FUNCTION_BLOCK FB_HVFAStorageSystem EXTENDS FB_SystemContinous
VAR_INPUT
	bLoadingAutomatic : BOOL; //variable to determine if storage is in loading mode
	aTelegramm_WMZ7x0 : ARRAY[1..cMBUS_MaxTelegrams] OF ST_MBus_Data2;
	aTelegramm_WMZx05 : ARRAY[1..cMBUS_MaxTelegrams] OF ST_MBus_Data2;
END_VAR
VAR_OUTPUT
	localState : ST_HVFAStorageState;
END_VAR
VAR
	{attribute 'OPC.UA.DA' := '1'}
	localSetParameters : ST_HVFAStorageSetParameters;
	
	//default parameters
	localDefaultParameters : ST_HVFAStorageSystemDefaultParameters;	

	//storage
	HVFAStorage : FB_HVFAStorage;
	
	//pumps
	PUx05 : FB_PumpGrundfosMagna3; //Magna 3 pump (network side)
	PU7x0 : FB_Pump2Point; //CM pump (storage side)

	//valves
	stSVx05DefaultParameters : ST_MixingValveDefaultParameters := (tTaskCycleTime := GlobalVariables.tCtrlCycleTime_MAIN, tCtrlCycleTime := GlobalVariables.tCtrlCycleTime_MAIN);
	stSVx06DefaultParameters : ST_MixingValveDefaultParameters := (tTaskCycleTime := GlobalVariables.tCtrlCycleTime_MAIN, tCtrlCycleTime := GlobalVariables.tCtrlCycleTime_MAIN);
	stRVx05DefaultParameters : ST_MixingValveDefaultParameters := (tTaskCycleTime := GlobalVariables.tCtrlCycleTime_MAIN, tCtrlCycleTime := GlobalVariables.tCtrlCycleTime_MAIN);
	
	SVx05 : FB_MixingValve := (ST_DefaultParameters := stSVx05DefaultParameters); //discrete inlet valve, valve motor needs continous signal but operates only between extreme positions
	SVx06 : FB_MixingValve := (ST_DefaultParameters := stSVx06DefaultParameters); //discrete outlet valve	, valve motor needs continous signal but operates only between extreme positions
	RVx05 : FB_MixingValve := (ST_DefaultParameters := stRVx05DefaultParameters); //continous mixing valve
	
	//sensors
	WMZ7x0 : FB_MollineC3HeatCounter;
	WMZx05 : FB_MollineC3HeatCounter;
	
	//internal variables
	bSetStatusOn_PUx05 : BOOL;
	bSetStatusOn_PU7x0 : BOOL;
	bSetStatusOn_SVx05 : BOOL;
	fSetPoint_SVx05 : REAL;
	bSetStatusOn_SVx06 : BOOL;
	fSetPoint_SVx06 : REAL;	
	bSetStatusOn_RVx05 : BOOL;
	fSetPoint_RVx05 : REAL;
	fExternalTemperature_RVx05 : REAL;
	nControlMode_RVx05 : E_MixingValveControlMode;
	bLoading : BOOL;
	
	//triggers
	SwitchToLoading : R_TRIG;
	SwitchToUnloading : F_TRIG;
	bFinishedSwitchMode : BOOL := TRUE;
END_VAR

//storage
HVFAStorage(localState => localState);

SelectLoadingMode();
SwitchToLoading(CLK := bLoading);
SwitchToUnloading(CLK := bLoading);

//MAIN must be called before SwitchMode to prevent pump signal chattering (signal is written after SwitchMode function), SwitchMode may only be called if system is on
MAIN();

//disrupt calling SystemFlowControl via MAIN() when mode is switched and call SwitchMode()
IF ((SwitchToLoading.Q OR SwitchToUnloading.Q) OR NOT bFinishedSwitchMode) AND bSetStatusOn THEN
	SwitchMode(bSwitchToLoading := bLoading,
		bFinishedSwitchMode => bFinishedSwitchMode);
END_IF;

//pumps
PUx05.GetState_Profibus();
PUx05(bSetStatusOnAutomatic := bSetStatusOn_PUx05,
	fSetPointAutomatic := 70,
	bAlgorithmPermission := bAlgorithmPermission,
	nControlModeAutomatic := 0);
PUx05.SetState_Profibus();

PU7x0(bSetStatusOnAutomatic := bSetStatusOn_PU7x0,
	bAlgorithmPermission := bAlgorithmPermission);
PU7x0.SetState_BO();

//valves
SVx05.GetState_AI();
SVx05(bSetStatusOnAutomatic := bSetStatusOn_SVx05,
	fSetPointAutomatic := fSetPoint_SVx05,
	bAlgorithmPermission := bAlgorithmPermission,
	nControlModeAutomatic := 0);
SVx05.SetState_AO();

SVx06.GetState_AI();
SVx06(bSetStatusOnAutomatic := bSetStatusOn_SVx06,
	fSetPointAutomatic := fSetPoint_SVx06,
	bAlgorithmPermission := bAlgorithmPermission,
	nControlModeAutomatic := 0);
SVx06.SetState_AO();

RVx05.GetState_AI();
RVx05(bSetStatusOnAutomatic := bSetStatusOn_RVx05,
	fSetPointAutomatic := fSetPoint,
	bAlgorithmPermission := bAlgorithmPermission,
	fTemperatureExternal := fExternalTemperature_RVx05,
	nControlModeAutomatic := 0);
RVx05.SetState_AO();

//insert heat counter telegramm from other task
WMZ7x0(aHeatCounterTelegramm := aTelegramm_WMZ7x0);
WMZx05(aHeatCounterTelegramm := aTelegramm_WMZx05);

IF bLoading = TRUE THEN
	fExternalTemperature_RVx05 := WMZ7x0.fReturnTemperazure;	
ELSE
	fExternalTemperature_RVx05 := WMZx05.fFeedTemperature;
END_IF

METHOD PROTECTED  CheckError : BOOL
VAR_INPUT
END_VAR
VAR_OUTPUT
	bError : BOOL;
END_VAR
VAR
	bError_PUx05 : BOOL;
END_VAR
//check for pump error
bError_PUx05 := PUx05.bError;
END_METHOD

METHOD PROTECTED  Operational : BOOL
VAR_INPUT
END_VAR
VAR_OUTPUT
	bSwitchToWorking : BOOL := FALSE;
END_VAR
//storage pump
bSetStatusOn_PU7x0 := TRUE;

//network pump
bSetStatusOn_PUx05 := TRUE;

//temperature controlling valve
bSetStatusOn_RVx05 := TRUE;

IF PUx05.bStatusOn THEN
	bSwitchToWorking := TRUE;
END_IF
END_METHOD

METHOD PROTECTED  RampDown : BOOL
VAR_INPUT
END_VAR
VAR_OUTPUT
	bRampDownFinished : BOOL := FALSE;
END_VAR
bSetStatusOn_PU7x0 := FALSE;
bSetStatusOn_PUx05 := FALSE;
bSetStatusOn_RVx05 := FALSE;

IF RVx05.fOperatingPoint<20 AND NOT PUx05.bStatusOn THEN
	bRampDownFinished := TRUE;
END_IF
END_METHOD

METHOD PROTECTED  RampUp : BOOL
VAR_INPUT
END_VAR
VAR_OUTPUT
	bRampUpFinished : BOOL := FALSE;
END_VAR
bSetStatusOn_SVx05 := TRUE;
bSetStatusOn_SVx06 := TRUE;

IF bLoading = TRUE THEN
	fSetPoint_SVx05 := 0;
	fSetPoint_SVx06 := 0;
	nControlMode_RVx05 := 2; //cooling mode (heats network)
	fExternalTemperature_RVx05 := WMZ7x0.fReturnTemperazure;	
	IF SVx05.fOperatingPoint<20 AND SVx06.fOperatingPoint<20 THEN
		bRampUpFinished := TRUE;
	END_IF
ELSE
	fSetPoint_SVx05 := 100;
	fSetPoint_SVx06 := 100;
	nControlMode_RVx05 := 1; //heating mode (cools network)
	fExternalTemperature_RVx05 := WMZx05.fFeedTemperature;
	IF SVx05.fOperatingPoint>80 AND SVx06.fOperatingPoint>80 THEN
		bRampUpFinished := TRUE;
	END_IF
END_IF
END_METHOD

METHOD PRIVATE SelectLoadingMode : BOOL
VAR_INPUT
END_VAR
IF control.bManualModeActivated THEN
	bLoading := localSetParameters.bLoadingManual;
ELSIF control.bAlgorithmModeActivated AND bAlgorithmPermission THEN
	bLoading := localSetParameters.bLoadingAlgorithm;
ELSE
	bLoading := bLoadingAutomatic;
END_IF
END_METHOD

METHOD PROTECTED   SetSetPointLimits : BOOL
VAR_INPUT
END_VAR
aSetPointLimits[1] := localDefaultParameters.aSetPointLimitsTemperature[1];
aSetPointLimits[2] := localDefaultParameters.aSetPointLimitsTemperature[2];
END_METHOD

METHOD PROTECTED  SetState : BOOL
VAR_INPUT
END_VAR
VAR_OUTPUT
END_VAR
fOperatingPoint := fExternalTemperature_RVx05;

controlState.bStatusOn := bSetStatusOn;
setPointState.aSetPointLimits := aSetPointLimits;
setPointState.fSetPoint := fSetPoint;
setPointState.fOperatingPoint := fOperatingPoint;
setPointState.sSetPointUnit := 'degreeC';
setPointState.sOperatingPointUnit := 'degreeC';
END_METHOD

PROPERTY ST_DefaultParameters : REFERENCE TO ST_HVFAStorageSystemDefaultParameters
SET
localDefaultParameters := ST_DefaultParameters;
END_SET
END_PROPERTY

METHOD PRIVATE SwitchMode : BOOL
VAR_INPUT
	bSwitchToLoading : BOOL; //if false switch to cooling
END_VAR
VAR_OUTPUT
	bFinishedSwitchMode : BOOL := FALSE;
END_VAR
VAR_INST
	bRampDownFinished : BOOL := FALSE;
END_VAR
//check system state
IF bRampDownFinished THEN
	IF bSwitchToLoading THEN
		fSetPoint_SVx05 := 0;
		fSetPoint_SVx06 := 0;
		nControlMode_RVx05 := 2; //cooling mode (heats network)	
		IF SVx05.fOperatingPoint<20 AND SVx06.fOperatingPoint<20 THEN
			//reset instant variable and switch on pump
			bRampDownFinished := FALSE;			
			bFinishedSwitchMode := TRUE;
			bSetStatusOn_PUx05 := TRUE;
		END_IF
		
	ELSE
		fSetPoint_SVx05 := 100;
		fSetPoint_SVx06 := 100;
		nControlMode_RVx05 := 1; //cooling mode (heats network)	
		IF SVx05.fOperatingPoint>80 AND SVx06.fOperatingPoint>80 THEN
			//reset instant variable and switch on pump
			bRampDownFinished := FALSE;			
			bFinishedSwitchMode := TRUE;
			bSetStatusOn_PUx05 := TRUE;
		END_IF
	END_IF
ELSE
	bSetStatusOn_PUx05 := FALSE;
	IF NOT PUx05.bStatusOn THEN
		bRampDownFinished := TRUE;
	END_IF
END_IF
END_METHOD

METHOD PROTECTED  Working : BOOL
VAR_INPUT
END_VAR
VAR_OUTPUT
	bSwitchToOperational : BOOL := FALSE;
END_VAR
//empty method
END_METHOD

END_FUNCTION_BLOCK

(* stored: Version 1.1.0.1, ProductVersion 3.1.4024.10
   POU FB_HVFAStorageSystem: Id {5fa1e97c-987f-49c1-82cf-2ddae1379d7b}, SpecialFunc None
   Method CheckError: Id {0a750c43-7566-4b1a-a185-b01eaf088ced}
   Method Operational: Id {38ce29c5-a9cb-42f6-b2da-f6e767b8efb9}
   Method RampDown: Id {035f2f79-06b9-4677-b822-1118600ad0da}
   Method RampUp: Id {0ce76782-d529-4b5d-8974-d96ba13ac874}
   Method SelectLoadingMode: Id {324f0df5-410b-4639-a772-5eb1aaf75a71}
   Method SetSetPointLimits: Id {f04c6bfe-2c3e-49d6-a8c4-445113c91ff8}
   Method SetState: Id {e91ff025-34ce-4425-84b2-ec422191accc}
   Property ST_DefaultParameters: Id {f1db4656-edfb-47d5-af6a-23dbe9289a24}
   Set Set: Id {293bdd0c-657e-4a38-8183-ebcb37193829}
   Method SwitchMode: Id {0eae4dfd-6df1-4d63-a8a7-6bb8ae2d2c72}
   Method Working: Id {c2454935-99da-4157-b03c-3bb74f66fa87} *)
